screen "Rad Settings" 1280x700, template "Navigation"
   TextField "Text field_15" at 511,20 size 403x43; Text 'RAD SETTINGS (uSv/h)'
   TextField "Text field_19" at 999,141 size 64x27; Text 'PUMP'
   TextField "Text field_20" at 1000,163 size 128x27; Text 'RAD LEVEL:'
   TextField "Text field_3" at 1003,201 size 83x27; Text 'VESSEL'
   TextField "Text field_4" at 1004,223 size 128x27; Text 'RAD LEVEL:'
   TextField "Text field_12" at 720,87 size 128x29; Text 'STATION 1'
   TextField "Text field_17" at 646,143 size 157x27; Text 'ALARM LEVEL:'
   IOField "I/O field_8" at 799,125 size 130x48; FormatPattern 9999.9
      ProcessValue <- "Station 1 Pump Rad Alarm Level"
   TextField "Text field_18" at 645,121 size 64x27; Text 'PUMP'
   IOField "I/O field_1" at 799,189 size 130x48; FormatPattern 9999.9
      ProcessValue <- "Station 1 Vessel Rad Alarm Level"
   TextField "Text field_1" at 646,207 size 157x27; Text 'ALARM LEVEL:'
   TextField "Text field_2" at 645,185 size 83x27; Text 'VESSEL'
   Group "Group_1" at 505,20 size 409x49; Text 'SYSTEM 1'
   IOField "I/O field_7" at 1132,207 size 130x48; FormatPattern 9999.9
      ProcessValue <- "Station 1 Vessel Rad Level"
   IOField "I/O field_9" at 1128,141 size 130x48; FormatPattern 9999.9
      ProcessValue <- "Station 1 Pump Rad Level"
   IOField "I/O field_2" at 1134,451 size 130x48; FormatPattern 9999.9
      ProcessValue <- "Waste Rad Level"
   TextField "Text field_7" at 1003,441 size 128x27; Text 'UNWANTED'
   TextField "Text field_8" at 1004,479 size 128x27; Text 'RAD LEVEL:'
   TextField "Text field_28" at 1063,108 size 128x29; Text 'STATION 1'
   Group "Group" at 999,141 size 129x49
   Group "Group_3" at 1003,201 size 129x49
   Group "Group_5" at 641,79 size 301x186
   IOField "I/O field_4" at 1132,368 size 130x48; FormatPattern 9999.9
      ProcessValue <- "Station 2 Vessel Rad Level"
   IOField "I/O field_6" at 1132,304 size 130x48; FormatPattern 9999.9
      ProcessValue <- "Station 2 Pump Rad Level"
   TextField "Text field_13" at 1003,301 size 64x27; Text 'PUMP'
   TextField "Text field_14" at 1004,323 size 128x27; Text 'RAD LEVEL:'
   TextField "Text field_22" at 1005,365 size 83x27; Text 'VESSEL'
   TextField "Text field_23" at 1006,387 size 128x27; Text 'RAD LEVEL:'
   TextField "Text field_24" at 1068,268 size 128x29; Text 'STATION 2'
   TextField "Text field_25" at 1015,71 size 228x29; Text 'FOR TESTING ONLY'
   Group "Group_7" at 642,275 size 301x186
   Group "Group_6" at 643,474 size 301x91
   TextField "Text field_27" at 1004,460 size 114x27; Text 'MATERIAL'
   IOField "I/O field_11" at 191,29 size 145x33; FormatPattern 9999.9; Unit  uSv/h
      ProcessValue <- "Station 1 Pump Rad Level"
   IOField "I/O field_12" at 191,71 size 152x33; FormatPattern 9999.9; Unit  uSv/h
      ProcessValue <- "Station 1 Vessel Rad Level"
   IOField "I/O field_14" at 191,110 size 146x33; FormatPattern 9999.9; Unit  uSv/h
      ProcessValue <- "Waste Rad Level"
   IOField "I/O field_23" at 193,149 size 150x33; FormatPattern 9999.9; Unit  uSv/h
      ProcessValue <- "Station 2 Pump Rad Level"
   IOField "I/O field_24" at 193,192 size 150x33; FormatPattern 9999.9; Unit  uSv/h
      ProcessValue <- "Station 2 Vessel Rad Level"
   Group "Group_28" at 293,236 size 117x42; Text 'SYSTEM 1'
   Group "Group_8" at 213,280 size 320x136; Picture "Graphic_1"
   Group "Group_9" at 213,428 size 320x137; Picture "Graphic_1"
   Group "Group_10" at 213,583 size 320x76; Picture "Graphic_1"
   Button "Template_Button_6" at 596,591 size 130x55; TextOff 'RAD SETTINGS'; Authorization "Maintenance"
      on Press: ActivateScreen("Rad Settings", 0)
      Visibility <- "CurrentGroupNum"
   Group "Group_12" at 958,551 size 315x121; TextOff 'RAD CTRL'; Text 'RINSE TO RAD LEVEL'; Authorization "Maintenance"; FormatPattern 9999
   Group "Group_14" at 366,71 size 315x121; TextOff 'RAD CTRL'; Text 'RINSE TO RAD LEVEL'; Authorization "Maintenance"; FormatPattern 9999
   IOField "I/O field_3" at 802,497 size 130x48; FormatPattern 9999.9
      ProcessValue <- "Waste Rad High Alarm"
   Group "Group_4" at 651,484 size 157x67
   TextField "Text field_6" at 652,484 size 128x27; Text 'UNWANTED'
   TextField "Text field_26" at 652,504 size 114x27; Text 'MATERIAL'
   TextField "Text field_5" at 651,524 size 157x27; Text 'ALARM LEVEL:'
   TextField "Text field_9" at 724,282 size 128x29; Text 'STATION 2'
   IOField "I/O field_5" at 801,322 size 130x48; FormatPattern 9999.9
      ProcessValue <- "Station 2 Pump Rad Alarm Level"
   IOField "I/O field_10" at 800,385 size 130x48; FormatPattern 9999.9
      ProcessValue <- "Station 2 Vessel Rad Alarm Level"
   TextField "Text field_16" at 647,403 size 157x27; Text 'ALARM LEVEL:'
   TextField "Text field_21" at 646,381 size 83x27; Text 'VESSEL'
   Group "Group_2" at 647,318 size 158x49
   TextField "Text field_11" at 647,318 size 64x27; Text 'PUMP'
   TextField "Text field_10" at 648,340 size 157x27; Text 'ALARM LEVEL:'
   TextField "Text field_29" at 305,236 size 94x39; Text 'ALMO'
   TextField "Text field_30" at 225,320 size 128x25; Text 'VESSEL CAVE'
   TextField "Text field_46" at 240,364 size 113x25; Text 'PUMP CAVE'
   TextField "Text field_49" at 275,283 size 120x27; Text 'STATION 1'
   TextField "Text field_50" at 390,282 size 88x27; Text '(uSv/h)'
   IOField "I/O field_13" at 355,315 size 113x34; FormatPattern 9999.9
      ProcessValue <- "Station 1 Vessel Rad Level"
   IOField "I/O field_15" at 355,359 size 113x34; FormatPattern 9999.9
      ProcessValue <- "Station 1 Pump Rad Level"
   GraphicView "Graphic view_2" at 476,313 size 36x36; Picture "Graphic_1"
      Visibility <- "Station 1 Vessel Rad Alarm"
   GraphicView "Graphic view_1" at 476,357 size 36x36; Picture "Graphic_1"
      Visibility <- "Station 1 Pump Rad Alarm"
   TextField "Text field_51" at 229,466 size 128x25; Text 'VESSEL CAVE'
   TextField "Text field_54" at 240,510 size 113x25; Text 'PUMP CAVE'
   TextField "Text field_57" at 273,431 size 120x27; Text 'STATION 2'
   TextField "Text field_58" at 388,430 size 88x27; Text '(uSv/h)'
   IOField "I/O field_16" at 353,462 size 112x34; FormatPattern 9999.9
      ProcessValue <- "Station 2 Vessel Rad Level"
   IOField "I/O field_17" at 353,507 size 112x34; FormatPattern 9999.9
      ProcessValue <- "Station 2 Pump Rad Level"
   GraphicView "Graphic view_6" at 473,460 size 36x36; Picture "Graphic_1"
      Visibility <- "Station 2 Vessel Rad Alarm"
   GraphicView "Graphic view_4" at 474,506 size 36x36; Picture "Graphic_1"
      Visibility <- "Station 2 Pump Rad Alarm"
   TextField "Text field_47" at 239,591 size 114x25; Text 'UNWANTED'
   IOField "I/O field_18" at 358,603 size 112x34; FormatPattern 9999.9
      ProcessValue <- "Waste Rad Level"
   GraphicView "Graphic view_3" at 476,601 size 36x36; Picture "Graphic_1"
      Visibility <- "Waste Rad Alarm"
   TextField "Text field_31" at 249,609 size 102x25; Text 'MATERIAL'
   TextField "Text field_32" at 279,627 size 66x25; Text 'VAULT'
   Group "Group_11" at 979,585 size 80x70; TextOff 'RAD CTRL'; Authorization "Maintenance"
   TextField "Text field_39" at 974,551 size 283x29; Text 'CONTROL TO RAD LEVEL'
   IOField "I/O field_19" at 1096,606 size 130x48; Authorization "Maintenance"; FormatPattern 9999.9
      ProcessValue <- "S1 Auto Rinse to RAD Level"
   TextField "Text field_40" at 1078,580 size 195x22; Text 'RAD LEVEL SP (uSv/h)'
   Button "Button_15" at 979,585 size 80x70; TextOff 'AUTO RAD CTRL'; Authorization "Maintenance"
      on Press: InvertBit("S1 Auto Use RAD CTRL")
   GraphicIOField "PlotLight_Round_GN_6" at 1033,587 size 22x23; PictureOn "PilotLight_Round_GN_On_256c"; PictureOff "PilotLight_Round_GN_Off_256c"; Authorization "Maintenance"
      ProcessValue <- "S1 Auto Use RAD CTRL"
   Group "Group_13" at 387,105 size 80x70; TextOff 'RAD CTRL'; Authorization "Maintenance"
   TextField "Text field_33" at 384,71 size 283x29; Text 'CONTROL TO RAD LEVEL'
   IOField "I/O field_20" at 504,126 size 130x48; Authorization "Maintenance"; FormatPattern 9999.9
      ProcessValue <- "S2 Auto Rinse to RAD Level"
   TextField "Text field_34" at 486,100 size 195x22; Text 'RAD LEVEL SP (uSv/h)'
   Button "Button_1" at 387,105 size 80x70; TextOff 'AUTO RAD CTRL'; Authorization "Maintenance"
      on Press: InvertBit("S2 Auto Use RAD CTRL")
   GraphicIOField "PlotLight_Round_GN_1" at 441,107 size 22x23; PictureOn "PilotLight_Round_GN_On_256c"; PictureOff "PilotLight_Round_GN_Off_256c"; Authorization "Maintenance"
      ProcessValue <- "S2 Auto Use RAD CTRL"

screen "Alarm Screen" 1280x700, template "Navigation"
   AlarmView "Alarm view_1" at 210,51 size 1021x325
   Group "Group_3" at 552,3 size 222x42; Text 'SYSTEM 1'
   AlarmView "Alarm view_2" at 211,416 size 1020x262
   TextField "Text field_1" at 239,386 size 210x34; Text 'ALARM BUFFER'
   TextField "Text field_13" at 557,3 size 210x39; Text 'ALARM VIEW'

screen "Status" 1280x700, template "Navigation"
   Group "Group_4" at 223,19 size 217x247
   Group "Group_3" at 1012,378 size 245x42; Text 'SYSTEM 1'
   Group "Group_2" at 1023,427 size 226x122; PictureOff "PilotLight_Round_G_Off_256c"; PictureOn "PilotLight_Round_R_On_256c"
   Group "Group_6" at 1023,555 size 226x122; PictureOff "PilotLight_Round_G_Off_256c"; PictureOn "PilotLight_Round_R_On_256c"
   Group "Group_8" at 192,279 size 261x74
   Group "Group_5" at 463,11 size 545x342
   Group "Group_9" at 1000,11 size 273x342
   Rectangle "Rectangle_9" at 1001,11 size 273x684
      Visibility <- "CurrentGroupNum"
   Button "Template_Button_3" at 246,85 size 166x69; TextOff 'S1 SETTINGS'
      on Press: function_efd93a16("Station 1 Settings", 180, 100, -1, -1, 1)
   Button "Template_Button_1" at 246,175 size 166x69; TextOff 'S2 SETTINGS'
      on Press: function_efd93a16("Station 2 Settings", 180, 100, -1, -1, 1)
   TextField "Text field_1" at 230,25 size 210x27; Text 'CURRENT PROCESS'
   TextField "Text field_2" at 270,45 size 111x27; Text 'SETTINGS'
   IOField "I/O field_1" at 707,96 size 128x48; FormatPattern 999.99
      ProcessValue <- "Station 1 Total Water Supply Volume"
   TextField "Text field_3" at 474,108 size 183x29; Text 'WATER SUPPLY'
   TextField "Text field_6" at 837,107 size 18x29; Text 'L'
   TextField "Text field_8" at 474,86 size 244x29; Text 'STATION 1 CURRENT'
   Button "Button_1" at 874,76 size 98x74; TextOff 'S1 H20 RESET'
      on Press: function_efd93a16("S1 Container Change", 680, 360, -1, -1, 1)
      ObjectEnable <- "Station 1 Process Running"
   IOField "I/O field_2" at 709,189 size 128x48; FormatPattern 999.99
      ProcessValue <- "Station 2 Total Water Supply Volume"
   TextField "Text field_4" at 476,201 size 183x29; Text 'WATER SUPPLY'
   TextField "Text field_5" at 476,179 size 244x29; Text 'STATION 2 CURRENT'
   Button "Button_2" at 876,169 size 98x74; TextOff 'S2 H20 RESET'
      on Press: function_efd93a16("S2 Container Change", 680, 360, -1, -1, 1)
      ObjectEnable <- "Station 2 Process Running"
   TextField "Text field_7" at 838,200 size 18x29; Text 'L'
   IOField "I/O field_3" at 708,281 size 128x48; FormatPattern 999.99
      ProcessValue <- "Total Waste Drum Volume"
   TextField "Text field_9" at 475,297 size 197x29; Text 'SUPPLY VOLUME'
   TextField "Text field_10" at 475,276 size 235x29; Text 'UM DRUM CURRENT'
   Button "Button_3" at 875,261 size 98x74; TextOff 'UM RESET'
      on Press: function_efd93a16("UM Container Change", 680, 360, -1, -1, 1)
   TextField "Text field_11" at 837,292 size 18x29; Text 'L'
   TextField "Text field_12" at 826,20 size 182x27; Text 'FOR CONTAINER'
   TextField "Text field_13" at 832,42 size 158x27; Text 'CHANGE ONLY'
   TextField "Text field_25" at 474,130 size 101x29; Text 'VOLUME'
   TextField "Text field_26" at 476,222 size 101x29; Text 'VOLUME'
   GraphicIOField "PlotLight_Round_R" at 1183,459 size 33x31; PictureOff "PilotLight_Round_G_Off_256c"; PictureOn "PilotLight_Round_R_On_256c"
      ProcessValue <- "Station 1 Pump Error Code Bit"
   TextField "Text field_16" at 1031,461 size 148x25; Text 'ERROR STATUS'
   TextField "Text field_17" at 1032,503 size 126x25; Text 'ERROR CODE'
   TextField "Text field_18" at 1085,430 size 120x27; Text 'STATION 1'
   IOField "I/O field_5" at 1170,499 size 60x34; FormatPattern 999
      ProcessValue <- "Station 1 Pump Error Code"
   TextField "Text field_22" at 1026,378 size 223x39; Text 'PUMP STATUS'
   GraphicIOField "PlotLight_Round_R_1" at 1183,587 size 33x31; PictureOn "PilotLight_Round_R_On_256c"; PictureOff "PilotLight_Round_G_Off_256c"
      ProcessValue <- "Station 2 Pump Error Code Bit"
   TextField "Text field_21" at 1031,589 size 148x25; Text 'ERROR STATUS'
   TextField "Text field_23" at 1032,631 size 126x25; Text 'ERROR CODE'
   TextField "Text field_24" at 1085,558 size 120x27; Text 'STATION 2'
   IOField "I/O field_4" at 1170,627 size 60x34; FormatPattern 999
      ProcessValue <- "Station 2 Pump Error Code"
   TextField "Text field_27" at 231,282 size 193x27; Text 'SYSTEM VERSION'
   IOField "I/O field_8" at 198,311 size 246x28; FormatPattern ????????????????????
      ProcessValue <- "System Version"
   IOField "I/O field_9" at 1011,96 size 128x48; FormatPattern 999.99
      ProcessValue <- "Station 1 Total Water Supply Update"
   TextField "Text field_28" at 1049,20 size 200x27; Text 'CORRECT VOLUME'
   TextField "Text field_29" at 1076,42 size 141x27; Text 'MAINT ONLY'
   TextField "Text field_30" at 1140,108 size 18x29; Text 'L'
   Button "Button_4" at 1164,75 size 98x74; TextOff 'S1 H20 UPDATE'
      on Press: SetBit("Station 1 Water Update")
      ObjectEnable <- "Station 1 Process Running"
   IOField "I/O field_10" at 1012,187 size 128x48; FormatPattern 999.99
      ProcessValue <- "Station 2 Total Water Supply Update"
   Button "Button_5" at 1164,169 size 98x74; TextOff 'S2 H20 UPDATE'
      on Press: SetBit("Station 2 Water Update")
      ObjectEnable <- "Station 2 Process Running"
   TextField "Text field_31" at 1139,201 size 18x29; Text 'L'
   IOField "I/O field_11" at 1012,279 size 128x48; FormatPattern 999.99
      ProcessValue <- "Total Waste Drum Update"
   TextField "Text field_32" at 1143,290 size 18x29; Text 'L'
   Button "Button_6" at 1164,261 size 98x74; TextOff 'UM UPDATE'
      on Press: SetBit("Waste Drum Update")

Template "Navigation" 1280x700
   Button "Template_Button_3" at 35,8 size 130x55; TextOff 'HOME'
      on Press: ActivateScreen("Home Screen", 0)
   Button "Template_Button_5" at 35,143 size 130x55; TextOff 'STATUS'
      on Press: ActivateScreen("Status", 0)
   Button "Template_Button_9" at 36,493 size 130x55; TextOff 'USER CONTROL'
      on Press: ActivateScreen("User Control", 0)
      Visibility <- "CurrentGroupNum"
   Button "Template_Button_4" at 35,75 size 130x55; TextOff 'ALARMS'
      on Press: ActivateScreen("Alarm Screen", 0)
   Rectangle "Template_Rectangle_1" at 27,209 size 147x272
      Visibility <- "CurrentGroupNum"
   Button "Template_Button_1" at 35,215 size 130x55; TextOff 'STATION 1 MANUAL'; Authorization "Maintenance"
      on Click: ActivateScreen("S1 Manual Mode", 0)
      Visibility <- "CurrentGroupNum"
   Button "Template_Button_2" at 35,351 size 130x55; TextOff 'STATION 1 SETUP'; Authorization "Maintenance"
      on Press: ActivateScreen("S1 Setup Screen", 0)
      Visibility <- "CurrentGroupNum"
   Button "Template_Button_7" at 35,419 size 130x55; TextOff 'STATION 2 SETUP'; Authorization "Maintenance"
      on Press: ActivateScreen("S2 Setup Screen", 0)
      Visibility <- "CurrentGroupNum"
   Button "Template_Button_8" at 35,283 size 130x55; TextOff 'STATION 2 MANUAL'; Authorization "Maintenance"
      on Press: ActivateScreen("S2 Manual Mode", 0)
      Visibility <- "CurrentGroupNum"

PopupScreen "Station 1 Settings" 1050x700
   TextField "Text field_15" at 199,16 size 372x43; Text 'STATION 1 SETTINGS'
   Button "Template_Button_3" at 37,480 size 166x69; TextOff 'RETURN'
      on Press: function_efd93a16()
   Group "Group_5" at 190,16 size 385x49; Text 'SYSTEM 1'
   Group "Group" at 34,91 size 275x295; Authorization "Maintenance"
   Group "Group_2" at 348,91 size 275x235; Authorization "Maintenance"
   Group "Group_7" at 661,32 size 275x164; Authorization "Maintenance"
   Group "Group_3" at 661,195 size 275x164; Authorization "Maintenance"
   Group "Group_4" at 661,358 size 275x164; Authorization "Maintenance"
   TextField "Text field_12" at 65,96 size 206x29; Text 'PROCESS TIMERS'
   TextField "Text field_16" at 39,314 size 129x27; Text 'TOTAL NUM'
   IOField "I/O field_7" at 162,319 size 130x48; Authorization "Maintenance"; FormatPattern 999
      ProcessValue <- "S1 Auto Number of Rinses"
   TextField "Text field_17" at 39,275 size 124x27; Text 'TIME (ms):'
   IOField "I/O field_8" at 161,256 size 130x48; Authorization "Maintenance"; FormatPattern 99999
      ProcessValue <- "S1 Auto Rinse Run Time"
   TextField "Text field_18" at 38,253 size 72x27; Text 'RINSE'
   IOField "I/O field_9" at 160,194 size 130x48; Authorization "Maintenance"; FormatPattern 99999
      ProcessValue <- "S1 Auto Drain Run Time"
   TextField "Text field_19" at 39,191 size 75x27; Text 'DRAIN'
   TextField "Text field_20" at 40,213 size 124x27; Text 'TIME (ms):'
   TextField "Text field_21" at 39,337 size 93x27; Text 'CYCLES:'
   IOField "I/O field_18" at 160,133 size 130x48; Authorization "Maintenance"; FormatPattern 99999
      ProcessValue <- "S1 Auto Remove Run Time"
   TextField "Text field_41" at 39,130 size 94x27; Text 'REMOVE'
   TextField "Text field_42" at 40,152 size 124x27; Text 'TIME (ms):'
   TextField "Text field_4" at 381,95 size 210x29; Text 'PUMP MAX SPEED'
   TextField "Text field_5" at 377,204 size 83x27; Text 'DRAIN:'
   IOField "I/O field_1" at 455,196 size 101x48; Authorization "Maintenance"; FormatPattern 999
      ProcessValue <- "S1 Auto Pump Drain Max Speed"
   TextField "Text field_6" at 378,269 size 80x27; Text 'RINSE:'
   IOField "I/O field_2" at 455,260 size 101x48; Authorization "Maintenance"; FormatPattern 999
      ProcessValue <- "S1 Auto Pump Rinse Max Speed"
   TextField "Text field_13" at 554,269 size 51x27; Text 'RPM'
   TextField "Text field_14" at 555,204 size 51x27; Text 'RPM'
   TextField "Text field_37" at 360,141 size 102x27; Text 'REMOVE:'
   IOField "I/O field_17" at 454,133 size 101x48; Authorization "Maintenance"; FormatPattern 999
      ProcessValue <- "S1 Auto Pump Remove Max Speed"
   TextField "Text field_38" at 554,141 size 51x27; Text 'RPM'
   TextField "Text field_43" at 713,36 size 174x29; Text 'REMOVE RAMP'
   TextField "Text field_49" at 675,80 size 124x27; Text 'NO. STEPS:'
   IOField "I/O field_19" at 792,72 size 128x48; Authorization "Maintenance"; FormatPattern 999
      ProcessValue <- "S1Auto Ramp Remove Step"
   TextField "Text field_50" at 674,141 size 124x27; Text 'TIME (ms):'
   IOField "I/O field_22" at 791,134 size 128x48; Authorization "Maintenance"; FormatPattern 99999
      ProcessValue <- "S1Auto Ramp Remove Time"
   TextField "Text field_1" at 724,199 size 154x29; Text 'DRAIN RAMP'
   TextField "Text field_7" at 674,243 size 124x27; Text 'NO. STEPS:'
   IOField "I/O field_3" at 791,235 size 128x48; Authorization "Maintenance"; FormatPattern 999
      ProcessValue <- "S1 Auto Ramp Drain Step"
   TextField "Text field_8" at 673,304 size 124x27; Text 'TIME (ms):'
   IOField "I/O field_4" at 790,297 size 128x48; Authorization "Maintenance"; FormatPattern 99999
      ProcessValue <- "S1 Auto Ramp Drain Time"
   TextField "Text field_9" at 728,362 size 150x29; Text 'RINSE RAMP'
   TextField "Text field_10" at 672,408 size 124x27; Text 'NO. STEPS:'
   IOField "I/O field_5" at 792,398 size 125x48; Authorization "Maintenance"; FormatPattern 999
      ProcessValue <- "S1 Auto Ramp Rinse Step"
   TextField "Text field_11" at 671,467 size 124x27; Text 'TIME (ms):'
   IOField "I/O field_6" at 793,460 size 125x48; Authorization "Maintenance"; FormatPattern 99999
      ProcessValue <- "S1 Auto Ramp Rinse Time"

PopupScreen "Station 2 Settings" 1050x700
   TextField "Text field_15" at 225,19 size 372x43; Text 'STATION 2 SETTINGS'
   Button "Template_Button_3" at 50,453 size 166x69; TextOff 'RETURN'
      on Press: function_efd93a16()
   Group "Group_1" at 216,19 size 381x49; Text 'SYSTEM 1'
   Group "Group_3" at 672,182 size 264x164; Text 'WASTE RAMP'; Authorization "Maintenance"
   Group "Group_4" at 672,345 size 265x164; Authorization "Maintenance"
   Group "Group" at 56,76 size 275x290; Authorization "Maintenance"
   Group "Group_2" at 370,76 size 275x227; Authorization "Maintenance"
   Group "Group_7" at 672,19 size 264x164; Authorization "Maintenance"
   TextField "Text field_1" at 737,186 size 154x29; Text 'DRAIN RAMP'
   TextField "Text field_7" at 677,230 size 124x27; Text 'NO. STEPS:'
   IOField "I/O field_3" at 794,222 size 128x48; Authorization "Maintenance"; FormatPattern 999
      ProcessValue <- "S2 Auto Ramp Drain Step"
   TextField "Text field_8" at 676,291 size 124x27; Text 'TIME (ms):'
   IOField "I/O field_4" at 793,284 size 128x48; Authorization "Maintenance"; FormatPattern 99999
      ProcessValue <- "S2 Auto Ramp Drain Time"
   TextField "Text field_9" at 739,349 size 150x29; Text 'RINSE RAMP'
   TextField "Text field_10" at 678,395 size 124x27; Text 'NO. STEPS:'
   IOField "I/O field_5" at 798,385 size 125x48; Authorization "Maintenance"; FormatPattern 999
      ProcessValue <- "S2 Auto Ramp Rinse Step"
   TextField "Text field_11" at 677,454 size 124x27; Text 'TIME (ms):'
   IOField "I/O field_6" at 799,447 size 125x48; Authorization "Maintenance"; FormatPattern 99999
      ProcessValue <- "S2 Auto Ramp Rinse Time"
   TextField "Text field_12" at 95,81 size 206x29; Text 'PROCESS TIMERS'
   TextField "Text field_16" at 61,299 size 129x27; Text 'TOTAL NUM'
   IOField "I/O field_7" at 184,304 size 130x48; Authorization "Maintenance"; FormatPattern 999
      ProcessValue <- "S2 Auto Number of Rinses"
   TextField "Text field_17" at 61,260 size 124x27; Text 'TIME (ms):'
   IOField "I/O field_8" at 183,241 size 130x48; Authorization "Maintenance"; FormatPattern 99999
      ProcessValue <- "S2 Auto Rinse Run Time"
   TextField "Text field_18" at 60,238 size 72x27; Text 'RINSE'
   IOField "I/O field_9" at 182,179 size 130x48; Authorization "Maintenance"; FormatPattern 99999
      ProcessValue <- "S2 Auto Drain Run Time"
   TextField "Text field_19" at 61,176 size 75x27; Text 'DRAIN'
   TextField "Text field_20" at 62,198 size 124x27; Text 'TIME (ms):'
   TextField "Text field_21" at 61,322 size 93x27; Text 'CYCLES:'
   IOField "I/O field_15" at 182,117 size 130x48; Authorization "Maintenance"; FormatPattern 99999
      ProcessValue <- "S2 Auto Remove Run Time"
   TextField "Text field_34" at 61,114 size 94x27; Text 'REMOVE'
   TextField "Text field_35" at 62,136 size 124x27; Text 'TIME (ms):'
   TextField "Text field_4" at 407,80 size 210x29; Text 'PUMP MAX SPEED'
   TextField "Text field_5" at 393,182 size 83x27; Text 'DRAIN:'
   IOField "I/O field_1" at 476,174 size 101x48; Authorization "Maintenance"; FormatPattern 999
      ProcessValue <- "S2 Auto Pump Drain Max Speed"
   TextField "Text field_6" at 398,243 size 80x27; Text 'RINSE:'
   IOField "I/O field_2" at 477,236 size 101x48; Authorization "Maintenance"; FormatPattern 999
      ProcessValue <- "S2 Auto Pump Rinse Max Speed"
   TextField "Text field_13" at 581,243 size 51x27; Text 'RPM'
   TextField "Text field_14" at 579,182 size 51x27; Text 'RPM'
   TextField "Text field_36" at 376,120 size 102x27; Text 'REMOVE:'
   IOField "I/O field_17" at 476,112 size 101x48; Authorization "Maintenance"; FormatPattern 999
      ProcessValue <- "S2 Auto Pump Remove Max Speed"
   TextField "Text field_37" at 579,120 size 51x27; Text 'RPM'
   TextField "Text field_38" at 726,23 size 174x29; Text 'REMOVE RAMP'
   TextField "Text field_41" at 677,67 size 124x27; Text 'NO. STEPS:'
   IOField "I/O field_18" at 794,59 size 128x48; Authorization "Maintenance"; FormatPattern 999
      ProcessValue <- "S2 Auto Ramp Remove Step"
   TextField "Text field_42" at 676,128 size 124x27; Text 'TIME (ms):'
   IOField "I/O field_19" at 793,121 size 128x48; Authorization "Maintenance"; FormatPattern 99999
      ProcessValue <- "S2 Auto Ramp Remove Time"

PopupScreen "S1 Container Change" 400x400
   Button "Template_Button_3" at 145,301 size 166x69; TextOff 'RETURN'
      on Press: function_efd93a16()
   TextField "Text field_1" at 31,42 size 330x29; Text 'Have you changed the water'
   TextField "Text field_2" at 36,65 size 318x29; Text 'container and wish to reset'
   TextField "Text field_3" at 82,159 size 86x47; Text 'YES:'
   Button "Button_1" at 178,145 size 98x74; TextOff 'RESET'
      on Press: SetBit("Station 1 New Water Container"); ActivateScreen("Status", 0)
      ObjectEnable <- "Station 1 Run State"
   TextField "Text field_4" at 70,314 size 70x43; Text 'NO:'
   TextField "Text field_5" at 27,88 size 349x29; Text 'the current container volume?'
   TextField "Text field_6" at 136,10 size 128x29; Text 'STATION 1'

PopupScreen "S2 Container Change" 400x400
   Button "Template_Button_3" at 145,301 size 166x69; TextOff 'RETURN'
      on Press: function_efd93a16()
   TextField "Text field_1" at 44,42 size 330x29; Text 'Have you changed the water'
   TextField "Text field_2" at 52,65 size 318x29; Text 'container and wish to reset'
   TextField "Text field_3" at 82,159 size 86x47; Text 'YES:'
   Button "Button_1" at 178,145 size 98x74; TextOff 'RESET'
      on Press: SetBit("Station 2 New Water Container"); ActivateScreen("Status", 0)
      ObjectEnable <- "Station 2 Run State"
   TextField "Text field_4" at 70,314 size 70x43; Text 'NO:'
   TextField "Text field_5" at 42,88 size 349x29; Text 'the current container volume?'
   TextField "Text field_6" at 136,10 size 128x29; Text 'STATION 2'

PopupScreen "UM Container Change" 400x400
   Button "Template_Button_3" at 145,301 size 166x69; TextOff 'RETURN'
      on Press: function_efd93a16()
   TextField "Text field_1" at 62,42 size 300x29; Text 'Have you changed the UM'
   TextField "Text field_2" at 57,65 size 318x29; Text 'container and wish to reset'
   TextField "Text field_3" at 82,159 size 86x47; Text 'YES:'
   Button "Button_1" at 178,145 size 98x74; TextOff 'RESET'
      on Press: SetBit("Station 1 New Waste Container"); SetBit("Station 2 New Waste Container"); ActivateScreen("Status", 0)
      ObjectEnable <- "Station 1 Run State"
   TextField "Text field_4" at 70,314 size 70x43; Text 'NO:'
   TextField "Text field_5" at 47,88 size 349x29; Text 'the current container volume?'
   TextField "Text field_6" at 80,10 size 264x29; Text 'UNWANTED MATERIAL'

VB script "TitleUpdater"
   Dim title
   Set title = HmiRuntime.Screens(0).ScreenItems("Screen title")
   title.Text = HmiRuntime.BaseScreenName

scheduled task "Get User Name"
   on Action: function_f41c6f6c("CurrentUserName"); function_e1ab61de("CurrentGroupNum")
*)